(* IEC 61131-3 sources: AXOpen/src/components.abstractions/ctrl/src/AxoRobotics, 6 files *)

(* ---- AxoRoboticsCoordinates.st ---- *)
NAMESPACE AXOpen.Components.Abstractions.Robotics
    TYPE AxoRoboticsCoordinates : STRUCT
            {#ix-set:AttributeName = "<#Coordinate X#>"}
            X : REAL;
            {#ix-set:AttributeName = "<#Coordinate Y#>"}
            Y : REAL;
            {#ix-set:AttributeName = "<#Coordinate Z#>"}
            Z : REAL;
            {#ix-set:AttributeName = "<#Coordinate Rx#>"}
            Rx : REAL;
            {#ix-set:AttributeName = "<#Coordinate Ry#>"}
            Ry : REAL;
            {#ix-set:AttributeName = "<#Coordinate Rz#>"}
            Rz : REAL;
        END_STRUCT;
    END_TYPE
END_NAMESPACE

(* ---- AxoRoboticsMovementsParams.st ---- *)
NAMESPACE AXOpen.Components.Abstractions.Robotics
    TYPE AxoRoboticsMovementsParams : STRUCT
            {#ix-set:AttributeName = "<#ActionNo#>"}
            ActionNo:BYTE;
            {#ix-set:AttributeName = "<#GlobalSpeed#>"}
            GlobalSpeed:BYTE;
            {#ix-set:AttributeName = "<#ToolNo#>"}
            ToolNo:BYTE;
            {#ix-set:AttributeName = "<#WorkobjectNo#>"}
            WorkobjectNo:BYTE;
            {#ix-set:AttributeName = "<#PointNo#>"}
            PointNo:BYTE;
            {#ix-set:AttributeName = "<#UserSpecSpeed1#>"}
            UserSpecSpeed1:INT;
            {#ix-set:AttributeName = "<#UserSpecSpeed2#>"}
            UserSpecSpeed2:INT;
            {#ix-set:AttributeName = "<#Coordinates#>"}
            Coordinates :AxoRoboticsCoordinates;
        END_STRUCT;
    END_TYPE
END_NAMESPACE

(* ---- eAxoRoboticsDistance.st ---- *)
NAMESPACE AXOpen.Components.Abstractions.Robotics
    TYPE PUBLIC
        eAxoRoboticsDistance :
        (
            X,
            Y,
            Z,
            XY,
            XZ,
            YZ,
            XYZ
        );
    END_TYPE
END_NAMESPACE

(* ---- eAxoRoboticsStopType.st ---- *)
NAMESPACE AXOpen.Components.Abstractions.Robotics
    TYPE PUBLIC
        eAxoRoboticsStopType :
        (
            Soft,
            Quick
        );
    END_TYPE
END_NAMESPACE

(* ---- IAxoRobotics.st ---- *)
USING AXOpen.Core;
NAMESPACE AXOpen.Components.Abstractions.Robotics
    INTERFACE PUBLIC IAxoRobotics
        METHOD StartAtMain : AXOpen.Core.IAxoTaskState  END_METHOD
        METHOD StartMotorsAndProgram : AXOpen.Core.IAxoTaskState  END_METHOD
        METHOD StartMovements  :   AXOpen.Core.IAxoTaskState
            VAR_IN_OUT
                inData : AxoRoboticsMovementsParams;
            END_VAR
        END_METHOD
        METHOD StopMovements  :   AXOpen.Core.IAxoTaskState
            VAR_INPUT
                inStopType : eAxoRoboticsStopType;
            END_VAR
        END_METHOD
        METHOD StopMovementsAndProgram  :   AXOpen.Core.IAxoTaskState
            VAR_INPUT
                inStopType : eAxoRoboticsStopType;
            END_VAR
        END_METHOD

    END_INTERFACE
END_NAMESPACE

(* ---- AxoRoboticsBasicCoordinates.st ---- *)
NAMESPACE AXOpen.Components.Abstractions.Robotics
    {S7.extern=ReadWrite}
    CLASS PUBLIC AxoRoboticsBasicCoordinates
        VAR PUBLIC
            {#ix-set:AttributeName = "<#Coordinate X#>"}
            X : REAL;
            {#ix-set:AttributeName = "<#Coordinate Y#>"}
            Y : REAL;
            {#ix-set:AttributeName = "<#Coordinate Z#>"}
            Z : REAL;
        END_VAR
    END_CLASS
END_NAMESPACE
